VAR_GLOBAL CONSTANT
	/// "Index-Group/Offset", GET_SYMHANDLE_BYNAME
	cGET_SYMHANDLE_BYNAME: UDINT := 16#F003;
	/// "Index-Group/Offset", READ_WRITE_SYMVAL_BYHANDLE
	cREAD_WRITE_SYMVAL_BYHANDLE: UDINT := 16#F005;
END_VAR

(* stored: Version 1.1.0.1, ProductVersion 3.1.4019.2
   GVL ADS_IndexGroup: Id {06e1f24a-87bb-47a4-8d8e-fc0192b1e43e} *)
